FUNCTION_BLOCK State_Levi_Dropdown
VAR_INPUT
	drive_status: ARRAY [0..23] OF UINT;
	drive_diagnostics: ARRAY [0..23] OF UINT;
	State : E_Levi_States;
	Force_feedback_value : ARRAY[0..23] OF INT;
END_VAR

VAR_OUTPUT
	Error: BOOL;
	Back_to_ready : E_Levi_States;
	Run_z_liftoff_calc : BOOL;
END_VAR

VAR_IN_OUT
	Control_word_array : ARRAY[0..23] OF UINT;
	drive_feedback_timeouts : ARRAY[0..23] OF UINT;
	force_values : ARRAY[0..11] OF INT;
	Drive_current_error : ARRAY[0..23] OF BOOL;
	error_specifics: ARRAY [0..23] OF Drive_error_mapping;
END_VAR

VAR
	current_dropdown : LREAL := -3; //A
	count_cycles: INT;
	n_drive_warnings: UINT;
	n_drive_errors: UINT;
	
	i: INT;
END_VAR

Run_z_liftoff_calc := FALSE;

Back_to_ready := E_Levi_States.LEVI_DROPDOWN;

FOR i:=0 TO 23 DO
	Control_word_array[i] := 16#E000;
END_FOR

(*
GVL_LEVI.Control_lat_parameters.blevi_operational := FALSE;
GVL_LEVI.Control_vert_parameters.blevi_operational := FALSE;
GVL_LEVI.FB_Control_lat.stlateral_levitation_control_P := GVL_LEVI.Control_lat_parameters;
GVL_LEVI.FB_Control_vert.stvertical_levitation_control_P := GVL_LEVI.Control_vert_parameters;
*)

//Check if there are errors
Error := Check_drives(drive_status := drive_status, 
					drive_diagnostics := drive_diagnostics, 
					drive_last_request_value := force_values,
					drive_last_feedback_value := Force_feedback_value,
					drive_feedback_timeouts := drive_feedback_timeouts,
					State := State,
					errors := error_specifics,
					Drive_current_error := Drive_current_error,
					n_warns => n_drive_warnings, 
					n_errors => n_drive_errors);


force_values[0] := LREAL_TO_INT((current_dropdown * 1000.0)/ GVL_LEVI.configured_peak_current_hems);
force_values[1] := LREAL_TO_INT((current_dropdown * 1000.0)/ GVL_LEVI.configured_peak_current_hems);

force_values[2] := LREAL_TO_INT((current_dropdown * 1000.0)/ GVL_LEVI.configured_peak_current_hems);
force_values[3] := LREAL_TO_INT((current_dropdown * 1000.0)/ GVL_LEVI.configured_peak_current_hems);

force_values[4] := LREAL_TO_INT((current_dropdown * 1000.0)/ GVL_LEVI.configured_peak_current_hems);
force_values[5] := LREAL_TO_INT((current_dropdown * 1000.0)/ GVL_LEVI.configured_peak_current_hems);

force_values[6] := LREAL_TO_INT((current_dropdown * 1000.0)/ GVL_LEVI.configured_peak_current_hems);
force_values[7] := LREAL_TO_INT((current_dropdown * 1000.0)/ GVL_LEVI.configured_peak_current_hems);

force_values[8] := 0;
force_values[9] := 0;

force_values[10] := 0;
force_values[11] := 0;

count_cycles := count_cycles + 1;

IF count_cycles > 1000 THEN
	count_cycles := 0;
	Back_to_ready := E_Levi_States.LEVI_READY;
END_IF

END_FUNCTION_BLOCK

(* stored: Version 1.1.0.1
   POU State_Levi_Dropdown: Id {2ad43b60-0717-4b07-88ee-06a40ca8fdd4}, SpecialFunc None *)
